TYPE ST_MaintParam :
STRUCT
	nChangeTool			: INT;
END_STRUCT
END_TYPE

(* stored: Version 1.1.0.1, ProductVersion 3.1.4022.10
   DUT ST_MaintParam: Id {e9e16f2b-156a-460f-ac5d-a2e8f2d97b69} *)
